//---------------------------------------------------------------------------------------------------------------
//
//  HAUD 2024.04.26
//
//  - APPLICATION
//    - explicit simple example PRG for setting up application
//      - no additional interfaces or encapsulations
//      - works dirEctly on GVL_XTS namespace Ctrl/State structs
//      - no error handling, reset application from start
//
//  - Application controls:
//    - XtsTransport
//      - GVL_XTS.TransportCtrl
//      - GVL_XTS.TransportState
//
//    - Xts Stations
//      - GVL_XTS.StationCtrl[]
//      - GVL_XTS.StationState[]
//      - see MAIN.StationParameterInit for XtsStation parameters.
//        - Intention: for developing a transport layer, 
//                      the station parameters are part of the XTS, 
//                      the application primarily handles handshakes with XtsStations
//
//  - Application
//    - 5 single XtsStations
//      - automated handshakes 
//      - process with TON
//      - static targets
//
//---------------------------------------------------------------------------------------------------------------
// This SOFTWARE is provided as an Exemple by THE PROVIDER "as is" and "with all faults." THE PROVIDER makes no 
// representations or warranties of any kind concerning the safety, suitability, lack of viruses, inaccuracies, 
// typographical errors, or other harmful components of this SOFTWARE. There are inherent dangers in the use of 
// any software, and you are solely responsible for determining whether this SOFTWARE is compatible with your 
// equipment and other software installed on your equipment. You are also solely responsible for the protection 
// of your equipment and backup of your data, and THE PROVIDER will not be liable for any damages you may suffer 
// in connection with using, modifying, or distributing this SOFTWARE.
//---------------------------------------------------------------------------------------------------------------
PROGRAM MAIN_APP
VAR
  eInit         : E_PROGRESS;
  bStart        : BOOL;   // XtsTransport is initialized, CAGroup is built, All movers are enabled, XtsStations are cleared, XtsTransport base position for all movers is commanded, XtsStations are handshaked with timer
  bReset        : BOOL;   // All Xts Stations are cleared, requires new start

  nXpu          : UINT;
  nStateError,
  nState        : ARRAY[1..MAX_XPU] OF UINT;   // state var for application

  tonProcess          : ARRAY[1..MAX_XPU] OF ARRAY[1..MAX_STATION] OF Tc2_Standard.TON;
  tProcess            : ARRAY[1..MAX_XPU] OF ARRAY[1..MAX_STATION] OF TIME;

  // work vars
  nStation      : ARRAY[1..MAX_XPU] OF UINT;
  nTarget       : ARRAY[1..MAX_XPU] OF ARRAY[1..MAX_STATION] OF UINT;  // contains target the station is sending the mover to, after process handshake was done

  JobResult     : ARRAY[1..MAX_XPU] OF E_PROGRESS;
END_VAR

//-----------------------------------------------------------------------------
// wait for initialization to be complete before work may start
//-----------------------------------------------------------------------------
IF NOT (Main.eInit = E_PROGRESS.PROGRESS_DONE)
THEN
  eInit                               := E_PROGRESS.PROGRESS_INIT;
  bReset                              := FALSE;
  bStart                              := FALSE;
  memset(ADR(nState), 0, SIZEOF(nState));
  RETURN;
END_IF
//-----------------------------------------------------------------------------
// fetch reset anytime
//-----------------------------------------------------------------------------
IF bReset
THEN
  bReset                              := FALSE;
  bStart                              := FALSE;
  FOR nXpu := 1 TO MAX_XPU
  DO
    nState[nXpu]                      := 9000;  // states for clearing XtsTransport
  END_FOR
END_IF

FOR nXpu := 1 TO MAX_XPU
DO
CASE nState[nXpu] 
OF
  0:                                  // first PLC cycle
    eInit                             := E_PROGRESS.PROGRESS_BUSY;
    nState[nXpu]                      := 1;

    FOR nStation[nXpu] := 1 TO MAX_STATION
    DO
      tProcess[nXpu][nStation[nXpu]]              := T#650MS;
      nTarget [nXpu][nStation[nXpu]]              := SEL(nStation[nXpu]<MAX_STATION, 1, nStation[nXpu]+1);
    END_FOR

  1:
    // do other init stuff here
    eInit                             := E_PROGRESS.PROGRESS_DONE;
    nState[nXpu]                      := 10;

  10:                                 // starts from here
    IF bStart
    THEN
      nStateError[nXpu]               := 0;
      nState[nXpu]                    := 100; // let's go
    END_IF
    
  100:                                // clear interface
    GVL_XTS.XtsTransportCtrl[nXpu].Cmd      := E_XTS_TRANSPORT_CTRL.CMD_NULL;
    nState[nXpu]                            := 110;

  110:                                // check initialization of XtsTransport, wait for either MoverDetection being valid or OperationMode.Simulation
    IF (GVL_XTS.XtsTransportState[nXpu].XpuInfo.IdDetectionValid) OR
       (GVL_XTS.XtsTransportState[nXpu].XpuInfo.OperationMode = OperationMode.Simulation)
    THEN
      // now XtsTransport is initialized, cyclic plausibility checks on Xpu are active
      nState[nXpu]                          := 120;
    END_IF

  120:                                // clear group for defined start situation
    GVL_XTS.XtsTransportCtrl[nXpu].Cmd      := E_XTS_TRANSPORT_CTRL.CMD_GROUP_CLEAR;

    IF (GVL_XTS.XtsTransportState[nXpu].State = E_XTS_TRANSPORT_STATE.TRANSPORT_GROUP_CLEAR + E_PROGRESS.PROGRESS_ERROR)
    THEN
      JobResult[nXpu]                       := GVL_XTS.CaGroupItf[nXpu].McResetAll(FALSE);
      nStateError[nXpu]                     := nState[nXpu];
      nState[nXpu]                          := 9011;

    ELSIF (GVL_XTS.XtsTransportState[nXpu].State = E_XTS_TRANSPORT_STATE.TRANSPORT_GROUP_CLEAR + E_PROGRESS.PROGRESS_DONE)
    THEN
      // CA Group is now in defined error free state
      nState[nXpu]                          := 130;
    END_IF

  130:                                // build Collision Avoidance group with all movers
    GVL_XTS.XtsTransportCtrl[nXpu].Cmd      := E_XTS_TRANSPORT_CTRL.CMD_GROUP_BUILD;

    IF (GVL_XTS.XtsTransportState[nXpu].State = E_XTS_TRANSPORT_STATE.TRANSPORT_GROUP_BUILD + E_PROGRESS.PROGRESS_ERROR)
    THEN
      JobResult[nXpu]                       := GVL_XTS.CaGroupItf[nXpu].McResetAll(FALSE);
      nStateError[nXpu]                     := nState[nXpu];
      nState[nXpu]                          := 9011;

    ELSIF (GVL_XTS.XtsTransportState[nXpu].State = E_XTS_TRANSPORT_STATE.TRANSPORT_GROUP_BUILD + E_PROGRESS.PROGRESS_DONE)
    THEN
      // CA Group contains all movers now
      // GVL_XTS.XtsTransportState.GroupInfo.AxisCount = MAX_MOVER
      nState[nXpu]                          := 140;
    END_IF

  140:                                // enable CA Group
    GVL_XTS.XtsTransportCtrl[nXpu].Cmd      := E_XTS_TRANSPORT_CTRL.CMD_GROUP_ENABLE;

    IF (GVL_XTS.XtsTransportState[nXpu].State = E_XTS_TRANSPORT_STATE.TRANSPORT_GROUP_ENABLE + E_PROGRESS.PROGRESS_ERROR)
    THEN
      JobResult[nXpu]                       := GVL_XTS.CaGroupItf[nXpu].McResetAll(FALSE);
      nStateError[nXpu]                     := nState[nXpu];
      nState[nXpu]                          := 9011;

    ELSIF (GVL_XTS.XtsTransportState[nXpu].State = E_XTS_TRANSPORT_STATE.TRANSPORT_GROUP_ENABLE + E_PROGRESS.PROGRESS_DONE)
    THEN
      // GVL_XTS.XtsTransportState.GroupInfo.CaGroupState = mcGroupStateNotReady
      nState[nXpu]                          := 150;
    END_IF

  150:                                // enable all movers
    GVL_XTS.XtsTransportCtrl[nXpu].Cmd      := E_XTS_TRANSPORT_CTRL.CMD_MOVER_ENABLE;

    IF (GVL_XTS.XtsTransportState[nXpu].State = E_XTS_TRANSPORT_STATE.TRANSPORT_MOVER_ENABLE + E_PROGRESS.PROGRESS_ERROR)
    THEN
      JobResult[nXpu]                       := GVL_XTS.CaGroupItf[nXpu].McResetAll(FALSE);
      nStateError[nXpu]                     := nState[nXpu];
      nState[nXpu]                          := 9011;

    ELSIF (GVL_XTS.XtsTransportState[nXpu].State = E_XTS_TRANSPORT_STATE.TRANSPORT_MOVER_ENABLE + E_PROGRESS.PROGRESS_DONE)
    THEN
      // GVL_XTS.XtsTransportState.GroupInfo.CaGroupState = mcGroupStateStandby
      nState[nXpu]                          := 160;
    END_IF

  160:                                // command all movers to startup position
    GVL_XTS.XtsTransportCtrl[nXpu].Cmd      := E_XTS_TRANSPORT_CTRL.CMD_TRANSPORT_START;

    IF (GVL_XTS.XtsTransportState[nXpu].State = E_XTS_TRANSPORT_STATE.TRANSPORT_START + E_PROGRESS.PROGRESS_DONE)
    THEN
      // all XtsStations are cleared
      // all movers are now waiting at GVL_XTS.XtsTransport.StartStationIndex
      // all movers are entered into GVL_XTS.StationList[GVL_XTS.XtsTransport.StartStationIndex]._stList 
      nState[nXpu]                          := 170;
    END_IF

  170:
    nState[nXpu]                            := 1000;

  1000:                               // automatic handshakes with XtsStations
    FOR nStation[nXpu] := 1 TO MAX_STATION
    DO
      CASE GVL_XTS.StationState[nXpu][nStation[nXpu]].eState
      OF
        E_STATION_STATE.STATION_DISABLE:          // switch on XtsStation
          GVL_XTS.StationCtrl[nXpu][nStation[nXpu]].eCmd      := E_STATION_CTRL.STATION_ENABLE;

        E_STATION_STATE.STATION_MOVER_ENTER:      // let mover enter
          // mover was detected in list and station is asking for mover entry
          GVL_XTS.StationCtrl[nXpu][nStation[nXpu]].eCmd      := E_STATION_CTRL.STATION_MOVER_ENTER;  // allow entry
          //GVL_XTS.StationCtrl[nStation].eCmd      := E_STATION_CTRL.STATION_MOVER_SEND;  // no process handshake, direct state change to MOVER_OUT 

        E_STATION_STATE.STATION_PROCESS_START:    // first process handshake, clear timer
          // mover has arrived and is in standstill, ready for process 
          tonProcess[nXpu][nStation[nXpu]](
                              IN                  :=FALSE, 
                              PT                  :=tProcess[nXpu][nStation[nXpu]]);
          GVL_XTS.StationCtrl[nXpu][nStation[nXpu]].eCmd      := E_STATION_CTRL.STATION_PROCESS_START;

        E_STATION_STATE.STATION_PROCESS_DONE:     // second process handshake, timer runs now
          tonProcess[nXpu][nStation[nXpu]](
                              IN                  :=TRUE, 
                              PT                  :=tProcess[nXpu][nStation[nXpu]]);
          IF tonProcess[nXpu][nStation[nXpu]].Q
          THEN
            GVL_XTS.StationCtrl[nXpu][nStation[nXpu]].eCmd    := E_STATION_CTRL.STATION_PROCESS_DONE;
          END_IF

        E_STATION_STATE.STATION_MOVER_OUT:        // station wants to send out mover
          // when sending out mover, the data on Ctrl struct is absolute important
          // before allowing the outfeed of the mover, the data on Ctrl struct must be entered correctly
          // Ctrl.nTargetStation allows for flexible mover transport, this is fully depending on you to make sense aside this example

          GVL_XTS.StationCtrl[nXpu][nStation[nXpu]].nTargetStation  := TO_USINT(nTarget[nXpu][nStation[nXpu]]); // static in this example
          GVL_XTS.StationCtrl[nXpu][nStation[nXpu]].nMask     := 2#1; // bitmask for mover ticket to next XtsStation; if you use more than one StopPos[] in XtsStation

          GVL_XTS.StationCtrl[nXpu][nStation[nXpu]].eCmd      := E_STATION_CTRL.STATION_MOVER_OUT;  // allow outfeed of mover

        E_STATION_STATE.STATION_MOVER_GONE:       // mover has travelled ReleaseDistance, XtsStation is now empty and ready for the next mover in queue
          GVL_XTS.StationCtrl[nXpu][nStation[nXpu]].nTargetStation  := 0;                           // clear target after mover left the station
          GVL_XTS.StationCtrl[nXpu][nStation[nXpu]].eCmd      := E_STATION_CTRL.STATION_MOVER_GONE; // last handshake for empty station
      END_CASE
    END_FOR


  9000:
    GVL_XTS.XtsTransportCtrl[nXpu].Cmd      := E_XTS_TRANSPORT_CTRL.CMD_NULL;
    nState[nXpu]                            := 9010;

  9010:                               // halt all movers and clear group
    GVL_XTS.XtsTransportCtrl[nXpu].Cmd      := E_XTS_TRANSPORT_CTRL.CMD_GROUP_CLEAR;

    IF (GVL_XTS.XtsTransportState[nXpu].State = E_XTS_TRANSPORT_STATE.TRANSPORT_GROUP_CLEAR + E_PROGRESS.PROGRESS_ERROR)
    THEN
      JobResult[nXpu]                       := GVL_XTS.CaGroupItf[nXpu].McResetAll(FALSE);
      nState[nXpu]                          := 9011;

    ELSIF (GVL_XTS.XtsTransportState[nXpu].State = E_XTS_TRANSPORT_STATE.TRANSPORT_GROUP_CLEAR + E_PROGRESS.PROGRESS_DONE)
    THEN
      // CA group cleared and mover in standstill
      nState[nXpu]                          := 9100;
    END_IF

  9011:
    JobResult[nXpu]                         := GVL_XTS.CaGroupItf[nXpu].McResetAll(TRUE);

    IF (JobResult[nXpu] = E_PROGRESS.PROGRESS_DONE)
    THEN
      nState[nXpu]                          := 9012;
      JobResult[nXpu]                       := GVL_XTS.CaGroupItf[nXpu].McResetAll(FALSE);
      JobResult[nXpu]                       := GVL_XTS.CaGroupItf[nXpu].Reset(FALSE);
    END_IF

  9012:
    JobResult[nXpu]                         := GVL_XTS.CaGroupItf[nXpu].Reset(TRUE);

    IF (JobResult[nXpu] = E_PROGRESS.PROGRESS_DONE)
    THEN
      nState[nXpu]                          := 9000;
      JobResult[nXpu]                       := GVL_XTS.CaGroupItf[nXpu].Reset(FALSE);
    END_IF


  9100:                               // switch off movers
    GVL_XTS.XtsTransportCtrl[nXpu].Cmd      := E_XTS_TRANSPORT_CTRL.CMD_MOVER_DISABLE;

    IF (GVL_XTS.XtsTransportState[nXpu].State >= E_XTS_TRANSPORT_STATE.TRANSPORT_MOVER_DISABLE + E_PROGRESS.PROGRESS_ERROR)
    THEN
      nState[nXpu]                          := 9200;
    END_IF

  9200:                               // clear All XtsStations
    nState[nXpu]                            := 9300;
    FOR nStation[nXpu] := 1 TO MAX_STATION
    DO
       GVL_XTS.StationCtrl[nXpu][nStation[nXpu]].eCmd      := E_STATION_CTRL.STATION_INIT;
    END_FOR

  9300:                               // disable All XtsStations
    nState[nXpu]                            := 10;   // go back to start
    FOR nStation[nXpu] := 1 TO MAX_STATION
    DO
       GVL_XTS.StationCtrl[nXpu][nStation[nXpu]].eCmd      := E_STATION_CTRL.STATION_DISABLE;
    END_FOR
END_CASE
END_FOR

END_PROGRAM

(* stored: Version 1.1.0.1, ProductVersion 3.1.4026.12
   POU MAIN_APP: Id {a42cfa77-97a5-4ec9-b576-fd1e63c4d66c}, SpecialFunc None *)
